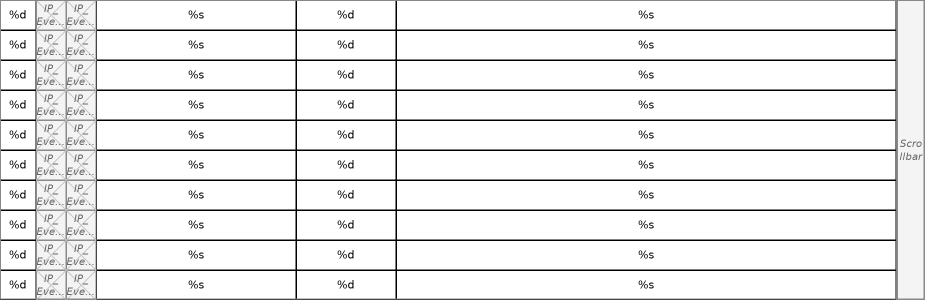
VISUALIZATION EventTable  // 925x300
VAR_IN_OUT
	data : ARRAY[1..512] OF ST_Event;
END_VAR
VAR 
	iIndex : INT;
END_VAR
    Group (0,0 896x30), invisible if: data[iIndex+1].iType = 0
        OnMouseClick: OpenDialog Dialog=SingleEvent, Parameters={data: data[iIndex+1]}, OpenModal=True, OpenCentered=True
        Rectangle (0,0 36x30), "%d", text variable: iIndex + 1
        Image (36,0 30x30), invisible if: data[iIndex+1].iType <> 1, image: IP_EventType.alarm
        Image (36,0 30x30), invisible if: data[iIndex+1].iType <> 2, image: IP_EventType.message
        Rectangle (96,0 200x30), "%s", text variable: LDT_TO_STRING(data[iIndex+1].iTimeStamp)
        Rectangle (296,0 100x30), "%d", text variable: data[iIndex+1].iEventId
        Image (66,0 30x30), invisible if: data[iIndex+1].eSeverity <> 4, image: IP_EventSeverity.critical
        Image (66,0 30x30), invisible if: data[iIndex+1].eSeverity <> 3, image: IP_EventSeverity.error
        Image (66,0 30x30), invisible if: data[iIndex+1].eSeverity <> 2, image: IP_EventSeverity.warning
        Image (66,0 30x30), invisible if: data[iIndex+1].eSeverity <> 1, image: IP_EventSeverity.info
        Image (66,0 30x30), invisible if: data[iIndex+1].eSeverity <> 0, image: IP_EventSeverity.verbose
        Rectangle (396,0 500x30), "%s", text variable: data[iIndex+1].sEventText
    Group (0,30 896x30), invisible if: data[iIndex+2].iType = 0
        OnMouseClick: OpenDialog Dialog=SingleEvent, Parameters={data: data[iIndex+2]}, OpenModal=True, OpenCentered=True
        Rectangle (0,0 36x30), "%d", text variable: iIndex + 2
        Image (36,0 30x30), invisible if: data[iIndex+2].iType <> 1, image: IP_EventType.alarm
        Image (36,0 30x30), invisible if: data[iIndex+2].iType <> 2, image: IP_EventType.message
        Rectangle (96,0 200x30), "%s", text variable: LDT_TO_STRING(data[iIndex+2].iTimeStamp)
        Rectangle (296,0 100x30), "%d", text variable: data[iIndex+2].iEventId
        Image (66,0 30x30), invisible if: data[iIndex+2].eSeverity <> 4, image: IP_EventSeverity.critical
        Image (66,0 30x30), invisible if: data[iIndex+2].eSeverity <> 3, image: IP_EventSeverity.error
        Image (66,0 30x30), invisible if: data[iIndex+2].eSeverity <> 2, image: IP_EventSeverity.warning
        Image (66,0 30x30), invisible if: data[iIndex+2].eSeverity <> 1, image: IP_EventSeverity.info
        Image (66,0 30x30), invisible if: data[iIndex+2].eSeverity <> 0, image: IP_EventSeverity.verbose
        Rectangle (396,0 500x30), "%s", text variable: data[iIndex+2].sEventText
    Group (0,60 896x30), invisible if: data[iIndex+3].iType = 0
        OnMouseClick: OpenDialog Dialog=SingleEvent, Parameters={data: data[iIndex+3]}, OpenModal=True, OpenCentered=True
        Rectangle (0,0 36x30), "%d", text variable: iIndex + 3
        Image (36,0 30x30), invisible if: data[iIndex+3].iType <> 1, image: IP_EventType.alarm
        Image (36,0 30x30), invisible if: data[iIndex+3].iType <> 2, image: IP_EventType.message
        Rectangle (96,0 200x30), "%s", text variable: LDT_TO_STRING(data[iIndex+3].iTimeStamp)
        Rectangle (296,0 100x30), "%d", text variable: data[iIndex+3].iEventId
        Image (66,0 30x30), invisible if: data[iIndex+3].eSeverity <> 4, image: IP_EventSeverity.critical
        Image (66,0 30x30), invisible if: data[iIndex+3].eSeverity <> 3, image: IP_EventSeverity.error
        Image (66,0 30x30), invisible if: data[iIndex+3].eSeverity <> 2, image: IP_EventSeverity.warning
        Image (66,0 30x30), invisible if: data[iIndex+3].eSeverity <> 1, image: IP_EventSeverity.info
        Image (66,0 30x30), invisible if: data[iIndex+3].eSeverity <> 0, image: IP_EventSeverity.verbose
        Rectangle (396,0 500x30), "%s", text variable: data[iIndex+3].sEventText
    Group (0,90 896x30), invisible if: data[iIndex+4].iType = 0
        OnMouseClick: OpenDialog Dialog=SingleEvent, Parameters={data: data[iIndex+4]}, OpenModal=True, OpenCentered=True
        Rectangle (0,0 36x30), "%d", text variable: iIndex + 4
        Image (36,0 30x30), invisible if: data[iIndex+4].iType <> 1, image: IP_EventType.alarm
        Image (36,0 30x30), invisible if: data[iIndex+4].iType <> 2, image: IP_EventType.message
        Rectangle (96,0 200x30), "%s", text variable: LDT_TO_STRING(data[iIndex+4].iTimeStamp)
        Rectangle (296,0 100x30), "%d", text variable: data[iIndex+4].iEventId
        Image (66,0 30x30), invisible if: data[iIndex+4].eSeverity <> 4, image: IP_EventSeverity.critical
        Image (66,0 30x30), invisible if: data[iIndex+4].eSeverity <> 3, image: IP_EventSeverity.error
        Image (66,0 30x30), invisible if: data[iIndex+4].eSeverity <> 2, image: IP_EventSeverity.warning
        Image (66,0 30x30), invisible if: data[iIndex+4].eSeverity <> 1, image: IP_EventSeverity.info
        Image (66,0 30x30), invisible if: data[iIndex+4].eSeverity <> 0, image: IP_EventSeverity.verbose
        Rectangle (396,0 500x30), "%s", text variable: data[iIndex+4].sEventText
    Group (0,120 896x30), invisible if: data[iIndex+5].iType = 0
        OnMouseClick: OpenDialog Dialog=SingleEvent, Parameters={data: data[iIndex+5]}, OpenModal=True, OpenCentered=True
        Rectangle (0,0 36x30), "%d", text variable: iIndex + 5
        Image (36,0 30x30), invisible if: data[iIndex+5].iType <> 1, image: IP_EventType.alarm
        Image (36,0 30x30), invisible if: data[iIndex+5].iType <> 2, image: IP_EventType.message
        Rectangle (96,0 200x30), "%s", text variable: LDT_TO_STRING(data[iIndex+5].iTimeStamp)
        Rectangle (296,0 100x30), "%d", text variable: data[iIndex+5].iEventId
        Image (66,0 30x30), invisible if: data[iIndex+5].eSeverity <> 4, image: IP_EventSeverity.critical
        Image (66,0 30x30), invisible if: data[iIndex+5].eSeverity <> 3, image: IP_EventSeverity.error
        Image (66,0 30x30), invisible if: data[iIndex+5].eSeverity <> 2, image: IP_EventSeverity.warning
        Image (66,0 30x30), invisible if: data[iIndex+5].eSeverity <> 1, image: IP_EventSeverity.info
        Image (66,0 30x30), invisible if: data[iIndex+5].eSeverity <> 0, image: IP_EventSeverity.verbose
        Rectangle (396,0 500x30), "%s", text variable: data[iIndex+5].sEventText
    Group (0,150 896x30), invisible if: data[iIndex+6].iType = 0
        OnMouseClick: OpenDialog Dialog=SingleEvent, Parameters={data: data[iIndex+6]}, OpenModal=True, OpenCentered=True
        Rectangle (0,0 36x30), "%d", text variable: iIndex + 6
        Image (36,0 30x30), invisible if: data[iIndex+6].iType <> 1, image: IP_EventType.alarm
        Image (36,0 30x30), invisible if: data[iIndex+6].iType <> 2, image: IP_EventType.message
        Rectangle (96,0 200x30), "%s", text variable: LDT_TO_STRING(data[iIndex+6].iTimeStamp)
        Rectangle (296,0 100x30), "%d", text variable: data[iIndex+6].iEventId
        Image (66,0 30x30), invisible if: data[iIndex+6].eSeverity <> 4, image: IP_EventSeverity.critical
        Image (66,0 30x30), invisible if: data[iIndex+6].eSeverity <> 3, image: IP_EventSeverity.error
        Image (66,0 30x30), invisible if: data[iIndex+6].eSeverity <> 2, image: IP_EventSeverity.warning
        Image (66,0 30x30), invisible if: data[iIndex+6].eSeverity <> 1, image: IP_EventSeverity.info
        Image (66,0 30x30), invisible if: data[iIndex+6].eSeverity <> 0, image: IP_EventSeverity.verbose
        Rectangle (396,0 500x30), "%s", text variable: data[iIndex+6].sEventText
    Group (0,180 896x30), invisible if: data[iIndex+7].iType = 0
        OnMouseClick: OpenDialog Dialog=SingleEvent, Parameters={data: data[iIndex+7]}, OpenModal=True, OpenCentered=True
        Rectangle (0,0 36x30), "%d", text variable: iIndex + 7
        Image (36,0 30x30), invisible if: data[iIndex+7].iType <> 1, image: IP_EventType.alarm
        Image (36,0 30x30), invisible if: data[iIndex+7].iType <> 2, image: IP_EventType.message
        Rectangle (96,0 200x30), "%s", text variable: LDT_TO_STRING(data[iIndex+7].iTimeStamp)
        Rectangle (296,0 100x30), "%d", text variable: data[iIndex+7].iEventId
        Image (66,0 30x30), invisible if: data[iIndex+7].eSeverity <> 4, image: IP_EventSeverity.critical
        Image (66,0 30x30), invisible if: data[iIndex+7].eSeverity <> 3, image: IP_EventSeverity.error
        Image (66,0 30x30), invisible if: data[iIndex+7].eSeverity <> 2, image: IP_EventSeverity.warning
        Image (66,0 30x30), invisible if: data[iIndex+7].eSeverity <> 1, image: IP_EventSeverity.info
        Image (66,0 30x30), invisible if: data[iIndex+7].eSeverity <> 0, image: IP_EventSeverity.verbose
        Rectangle (396,0 500x30), "%s", text variable: data[iIndex+7].sEventText
    Group (0,210 896x30), invisible if: data[iIndex+8].iType = 0
        OnMouseClick: OpenDialog Dialog=SingleEvent, Parameters={data: data[iIndex+8]}, OpenModal=True, OpenCentered=True
        Rectangle (0,0 36x30), "%d", text variable: iIndex + 8
        Image (36,0 30x30), invisible if: data[iIndex+8].iType <> 1, image: IP_EventType.alarm
        Image (36,0 30x30), invisible if: data[iIndex+8].iType <> 2, image: IP_EventType.message
        Rectangle (96,0 200x30), "%s", text variable: LDT_TO_STRING(data[iIndex+8].iTimeStamp)
        Rectangle (296,0 100x30), "%d", text variable: data[iIndex+8].iEventId
        Image (66,0 30x30), invisible if: data[iIndex+8].eSeverity <> 4, image: IP_EventSeverity.critical
        Image (66,0 30x30), invisible if: data[iIndex+8].eSeverity <> 3, image: IP_EventSeverity.error
        Image (66,0 30x30), invisible if: data[iIndex+8].eSeverity <> 2, image: IP_EventSeverity.warning
        Image (66,0 30x30), invisible if: data[iIndex+8].eSeverity <> 1, image: IP_EventSeverity.info
        Image (66,0 30x30), invisible if: data[iIndex+8].eSeverity <> 0, image: IP_EventSeverity.verbose
        Rectangle (396,0 500x30), "%s", text variable: data[iIndex+8].sEventText
    Group (0,240 896x30), invisible if: data[iIndex+9].iType = 0
        OnMouseClick: OpenDialog Dialog=SingleEvent, Parameters={data: data[iIndex+9]}, OpenModal=True, OpenCentered=True
        Rectangle (0,0 36x30), "%d", text variable: iIndex + 9
        Image (36,0 30x30), invisible if: data[iIndex+9].iType <> 1, image: IP_EventType.alarm
        Image (36,0 30x30), invisible if: data[iIndex+9].iType <> 2, image: IP_EventType.message
        Rectangle (96,0 200x30), "%s", text variable: LDT_TO_STRING(data[iIndex+9].iTimeStamp)
        Rectangle (296,0 100x30), "%d", text variable: data[iIndex+9].iEventId
        Image (66,0 30x30), invisible if: data[iIndex+9].eSeverity <> 4, image: IP_EventSeverity.critical
        Image (66,0 30x30), invisible if: data[iIndex+9].eSeverity <> 3, image: IP_EventSeverity.error
        Image (66,0 30x30), invisible if: data[iIndex+9].eSeverity <> 2, image: IP_EventSeverity.warning
        Image (66,0 30x30), invisible if: data[iIndex+9].eSeverity <> 1, image: IP_EventSeverity.info
        Image (66,0 30x30), invisible if: data[iIndex+9].eSeverity <> 0, image: IP_EventSeverity.verbose
        Rectangle (396,0 500x30), "%s", text variable: data[iIndex+9].sEventText
    Group (0,270 896x30), invisible if: data[iIndex+10].iType = 0
        OnMouseClick: OpenDialog Dialog=SingleEvent, Parameters={data: data[iIndex+10]}, OpenModal=True, OpenCentered=True
        Rectangle (0,0 36x30), "%d", text variable: iIndex + 10
        Image (36,0 30x30), invisible if: data[iIndex+10].iType <> 1, image: IP_EventType.alarm
        Image (36,0 30x30), invisible if: data[iIndex+10].iType <> 2, image: IP_EventType.message
        Rectangle (96,0 200x30), "%s", text variable: LDT_TO_STRING(data[iIndex+10].iTimeStamp)
        Rectangle (296,0 100x30), "%d", text variable: data[iIndex+10].iEventId
        Image (66,0 30x30), invisible if: data[iIndex+10].eSeverity <> 4, image: IP_EventSeverity.critical
        Image (66,0 30x30), invisible if: data[iIndex+10].eSeverity <> 3, image: IP_EventSeverity.error
        Image (66,0 30x30), invisible if: data[iIndex+10].eSeverity <> 2, image: IP_EventSeverity.warning
        Image (66,0 30x30), invisible if: data[iIndex+10].eSeverity <> 1, image: IP_EventSeverity.info
        Image (66,0 30x30), invisible if: data[iIndex+10].eSeverity <> 0, image: IP_EventSeverity.verbose
        Rectangle (396,0 500x30), "%s", text variable: data[iIndex+10].sEventText
    Scrollbar (897,0 28x300)
        p2245068023: GVL.iMAX_EVENTS - 10
        p1057716461: iIndex
END_VISUALIZATION

(* stored: Version 1.1.0.1, ProductVersion 3.1.4024.12
   Visu EventTable: Id {63974322-1e66-4922-bfa7-3b3ad08a4f63} *)
